PROGRAM task4
VAR
	sensor1 : SensorBrands;
END_VAR

sensor1 := SensorBrands.Parker;

END_PROGRAM

(* stored: Version 1.1.0.1, ProductVersion 3.1.4024.12
   POU task4: Id {aceb53d0-0c79-46ab-b12d-4a8988e85ed3}, SpecialFunc None *)
